{attribute 'GeneratedUsingTerminal: AMP8000-0030-0103-0103'}
{attribute addProperty BoxType "AMP8000-0030-0103-0103"}
{attribute addProperty Id "FSOEAT %Q*FSOE_6A82EB9321"}
{attribute addProperty CRC "1896473840"}
{attribute addProperty Size "21"}
TYPE FSoE_Slave_Connection_1_Master_Message_7109E4F0 EXTENDS OutputBase_10CEE7DE :
STRUCT
	{attribute addProperty Name "FSOE"}
	FSOE AT %Q* : FSOE_6A82EB93;
END_STRUCT
END_TYPE

(* stored: Version 1.2.0.0, ProductVersion 3.1.4024.11
   DUT FSoE_Slave_Connection_1_Master_Message_7109E4F0: Id {fbe1c46a-5377-4839-a55e-5d8cc26ee97a} *)
